INTERFACE I_Command

METHOD PUBLIC Abort
VAR_INPUT
END_VAR
END_METHOD

METHOD PUBLIC Execute
END_METHOD

PROPERTY PUBLIC Feedback : I_CommandFeedback
GET
END_GET
END_PROPERTY

END_INTERFACE

(* stored: Version 1.1.0.1, ProductVersion 3.1.4024.11
   Itf I_Command: Id {c2374356-39d9-4a81-82d4-a9dd89072af4}
   Method Abort: Id {9525fb97-a63b-4487-bfa0-a5ee9240133e}
   Method Execute: Id {680cb84f-e285-4414-bb7d-46c7f81f4e85}
   Property Feedback: Id {bbcfb8ff-ca21-4b29-a60f-53e7766a1ef8}
   Get Get: Id {8fb8f332-b019-4000-bfc6-c905c9bc84f1} *)
